(* PLC project SafeLOGIC-1, BrAutomation SafeDESIGNER  4.4.0.0 *)
(* stored: companyURL http://www.br-automation.com, creationDateTime Mon Oct 25 15:15:50 2021 *)

PROGRAM Main
  VAR  (* added by the conversion: wires and edge detectors of the diagram *)
    _AND_S57_OUT : ANY;
    _SAFEBOOL_TO_BOOL24_OUT : BOOL;
  END_VAR

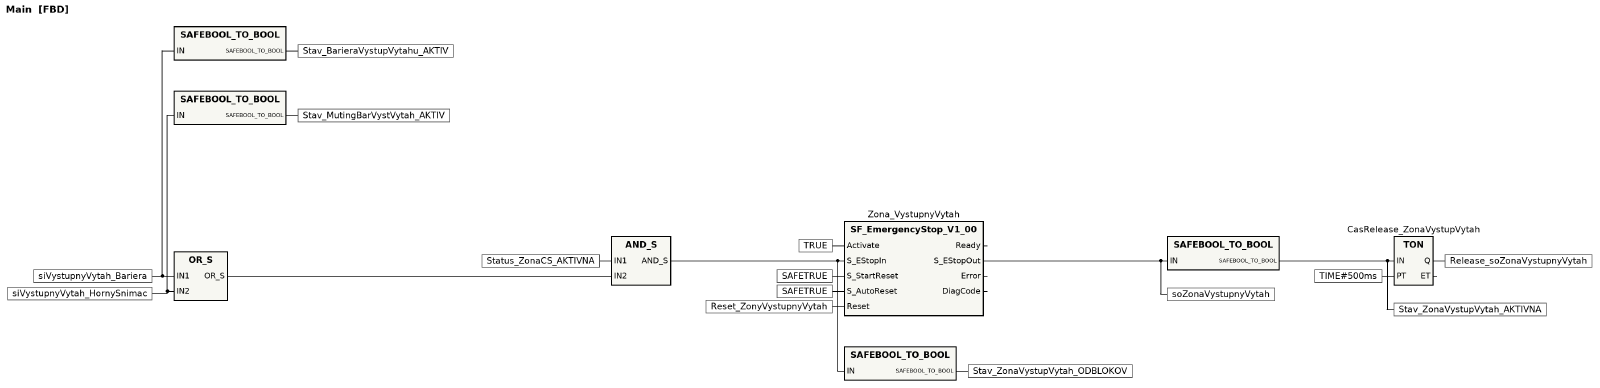
(* FBD diagram, written out as Structured Text *)
_AND_S57_OUT := AND_S(Status_ZonaCS_AKTIVNA, OR_S(siVystupnyVytah_Bariera, siVystupnyVytah_HornySnimac));
Zona_VystupnyVytah(Activate := TRUE, S_EStopIn := _AND_S57_OUT, S_StartReset := SAFETRUE, S_AutoReset := SAFETRUE, Reset := Reset_ZonyVystupnyVytah);
soZonaVystupnyVytah := Zona_VystupnyVytah.S_EStopOut;
_SAFEBOOL_TO_BOOL24_OUT := SAFEBOOL_TO_BOOL(Zona_VystupnyVytah.S_EStopOut);
CasRelease_ZonaVystupVytah(IN := _SAFEBOOL_TO_BOOL24_OUT, PT := TIME#500ms);
Release_soZonaVystupnyVytah := CasRelease_ZonaVystupVytah.Q;
Stav_BarieraVystupVytahu_AKTIV := SAFEBOOL_TO_BOOL(siVystupnyVytah_Bariera);
Stav_ZonaVystupVytah_ODBLOKOV := SAFEBOOL_TO_BOOL(_AND_S57_OUT);
Stav_MutingBarVystVytah_AKTIV := SAFEBOOL_TO_BOOL(siVystupnyVytah_HornySnimac);
Stav_ZonaVystupVytah_AKTIVNA := _SAFEBOOL_TO_BOOL24_OUT;
END_PROGRAM
